// TIA Portal project "赛题3" (V16)

(* hardware
DEVICE "S7-1200 station_2"  S7-1200 Station
   slot 0: "Rack_0"  S7-1200 Rack  Rack  V1.0
   slot 1: "PLC_1"  CPU 1214C DC/DC/DC  6ES7 214-1AG40-0XB0  V4.4
*)

// ===== PLC "PLC_1"  CPU 1214C DC/DC/DC =====

VAR_GLOBAL   // PLC tag table "默认变量表"
   "启动点" AT %M0.0 : Bool;
   "中间点1" AT %M0.1 : Bool;
   "中间点2" AT %M0.2 : Bool;
   "中间点3" AT %M0.3 : Bool;
   "中间点4" AT %M0.4 : Bool;
   "中间点5" AT %M1.0 : Bool;
   "车道绿灯" AT %Q0.0 : Bool;
   "车道黄灯" AT %Q0.1 : Bool;
   "车道红灯" AT %Q0.2 : Bool;
   "内部点1" AT %M2.0 : Bool;
   "内部点2" AT %M3.0 : Bool;
   "内部点3" AT %M4.0 : Bool;
   "内部点4" AT %M5.0 : Bool;
   "人道绿灯" AT %Q0.3 : Bool;
   "人道红灯" AT %Q0.4 : Bool;
   "Tag_1" AT %M9.0 : Bool;
   "Tag_2" AT %M9.1 : Bool;
   "Tag_3" AT %M9.2 : Bool;
   "Tag_4" AT %M6.0 : Bool;
END_VAR

// folder: System blocks/Program resources

DATA_BLOCK "IEC_Timer_0_DB0"   // DB1
{ S7_Optimized_Access := 'TRUE' }
AUTHOR : Simatic
FAMILY : IEC
NAME : IEC_TMR
VERSION : 1.0
// stored: InstanceOfName IEC_TIMER
"IEC_TIMER"
BEGIN
END_DATA_BLOCK

DATA_BLOCK "IEC_Timer_0_DB1"   // DB2
{ S7_Optimized_Access := 'TRUE' }
AUTHOR : Simatic
FAMILY : IEC
NAME : IEC_TMR
VERSION : 1.0
// stored: InstanceOfName IEC_TIMER
"IEC_TIMER"
BEGIN
END_DATA_BLOCK

DATA_BLOCK "IEC_Timer_0_DB2"   // DB3
{ S7_Optimized_Access := 'TRUE' }
AUTHOR : Simatic
FAMILY : IEC
NAME : IEC_TMR
VERSION : 1.0
// stored: InstanceOfName IEC_TIMER
"IEC_TIMER"
BEGIN
END_DATA_BLOCK

DATA_BLOCK "IEC_Timer_0_DB"   // DB4
{ S7_Optimized_Access := 'TRUE' }
AUTHOR : Simatic
FAMILY : IEC
NAME : IEC_TMR
VERSION : 1.0
// stored: InstanceOfName IEC_TIMER
"IEC_TIMER"
BEGIN
END_DATA_BLOCK

DATA_BLOCK "IEC_Timer_0_DB_1"   // DB5
{ S7_Optimized_Access := 'TRUE' }
AUTHOR : Simatic
FAMILY : IEC
NAME : IEC_TMR
VERSION : 1.0
// stored: InstanceOfName IEC_TIMER
"IEC_TIMER"
BEGIN
END_DATA_BLOCK

DATA_BLOCK "IEC_Timer_0_DB_2"   // DB6
{ S7_Optimized_Access := 'TRUE' }
AUTHOR : Simatic
FAMILY : IEC
NAME : IEC_TMR
VERSION : 1.0
// stored: InstanceOfName IEC_TIMER
"IEC_TIMER"
BEGIN
END_DATA_BLOCK

// folder: (top level)

FUNCTION "块_1" : Void   // FC1, LAD
{ S7_Optimized_Access := 'TRUE' }
VERSION : 0.1
   VAR_INPUT
      start : Bool;
      G_X : Bool;
      Y_X : Bool;
      R_X : Bool;
   END_VAR
   VAR_OUTPUT
      C_green : Bool;
      C_red : Bool;
      C_yellow : Bool;
      R_green : Bool;
      R_red : Bool;
   END_VAR
   VAR_TEMP   // added for the SCL form of the ladder/FBD networks
      _w1 : Bool;
      _w2 : Bool;
   END_VAR
BEGIN

REGION Network 1
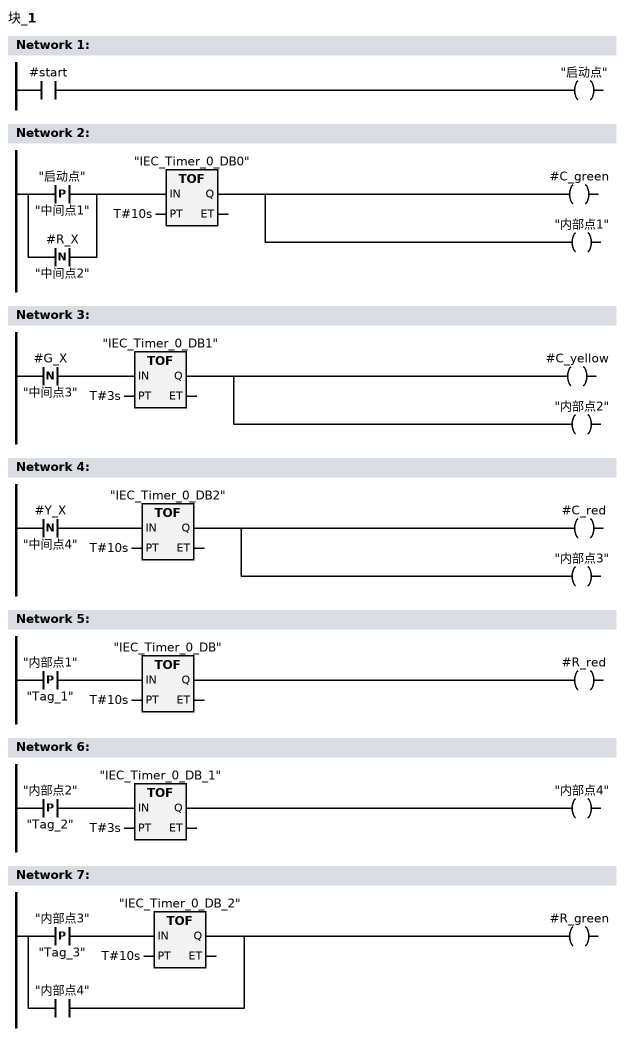
   RUNG wire#powerrail
      Contact( #start )
      Coil( "启动点" )
   END_RUNG
   // the same network as SCL:
   "启动点" := #start;
END_REGION

REGION Network 2
   #_w1 := "启动点" AND NOT "中间点1";   // rising edge of "启动点"
   "中间点1" := "启动点";
   #_w2 := NOT #R_X AND "中间点2";   // falling edge of #R_X
   "中间点2" := #R_X;
   "IEC_Timer_0_DB0".TOF(IN := #_w1 OR #_w2, PT := T#10s);
   #C_green := "IEC_Timer_0_DB0".Q;
   "内部点1" := "IEC_Timer_0_DB0".Q;
END_REGION

REGION Network 3
   #_w1 := NOT #G_X AND "中间点3";   // falling edge of #G_X
   "中间点3" := #G_X;
   "IEC_Timer_0_DB1".TOF(IN := #_w1, PT := T#3s);
   #C_yellow := "IEC_Timer_0_DB1".Q;
   "内部点2" := "IEC_Timer_0_DB1".Q;
END_REGION

REGION Network 4
   #_w1 := NOT #Y_X AND "中间点4";   // falling edge of #Y_X
   "中间点4" := #Y_X;
   "IEC_Timer_0_DB2".TOF(IN := #_w1, PT := T#10s);
   #C_red := "IEC_Timer_0_DB2".Q;
   "内部点3" := "IEC_Timer_0_DB2".Q;
END_REGION

REGION Network 5
   #_w1 := "内部点1" AND NOT "Tag_1";   // rising edge of "内部点1"
   "Tag_1" := "内部点1";
   "IEC_Timer_0_DB".TOF(IN := #_w1, PT := T#10s);
   #R_red := "IEC_Timer_0_DB".Q;
END_REGION

REGION Network 6
   #_w1 := "内部点2" AND NOT "Tag_2";   // rising edge of "内部点2"
   "Tag_2" := "内部点2";
   "IEC_Timer_0_DB_1".TOF(IN := #_w1, PT := T#3s);
   "内部点4" := "IEC_Timer_0_DB_1".Q;
END_REGION

REGION Network 7
   #_w1 := "内部点3" AND NOT "Tag_3";   // rising edge of "内部点3"
   "Tag_3" := "内部点3";
   "IEC_Timer_0_DB_2".TOF(IN := #_w1, PT := T#10s);
   #R_green := "IEC_Timer_0_DB_2".Q OR "内部点4";
END_REGION
END_FUNCTION

ORGANIZATION_BLOCK "Main"   // OB1, LAD, ProgramCycle
TITLE = "Main Program Sweep (Cycle)"
{ S7_Optimized_Access := 'TRUE' }
VERSION : 0.1
   VAR_INPUT
      Initial_Call : Bool;   // Initial call of this OB
      Remanence : Bool;   // =True, if remanent data are available
   END_VAR
BEGIN

REGION Network 1
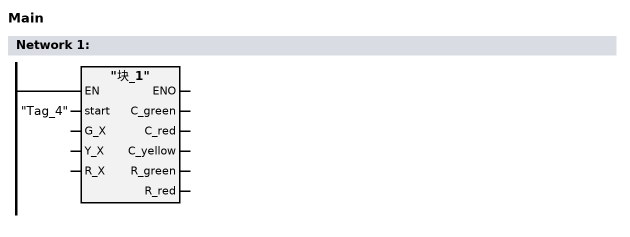
   RUNG wire#powerrail
      "块_1"(start := "Tag_4", G_X :=, Y_X :=, R_X :=, C_green =>, C_red =>, C_yellow =>, R_green =>, R_red =>)
   END_RUNG
   // the same network as SCL:
   "块_1"(start := "Tag_4");
END_REGION
END_ORGANIZATION_BLOCK